# B&R Automation Studio project PO_automation
Automation Studio 4.5.2.102

## Configuration Config1

### Task classes (Cpu.sw)
```
Cyclic#1:
  Program <- Program.prg
Binaries: udbdef, TCData, ashwd, User, asfw, arconfig, sysconf, Role, ashwac, iomap
Libraries: library
```

## Logical view

Binary libraries used (declarations not repeated): operator, runtime, astime, AsIecCon

### Global.var
```iecst
VAR
	fb_controller : FB_Regulator;
	speed : REAL;
	counter : UINT;
	enable : BOOL;
	fb_motor2 : FB_Motor;
	fb_motor1 : FB_Motor;
END_VAR
```

### Library Logical/Libraries/library (ANSIC)

#### FB_Integrator.c
```c
#include <bur/plctypes.h>
#ifdef __cplusplus
	extern "C"
	{
#endif
	#include "library.h"
#ifdef __cplusplus
	};
#endif
/* TODO: Add your comment here */
void FB_Integrator(struct FB_Integrator* inst)
{
	/*TODO: Add your code here*/
	inst->out = inst->dt * inst->in + inst->prev_value;
	inst->prev_value = inst->out;
}
```

#### library.fun - Exported functions and function blocks
```iecst
{REDUND_ERROR} FUNCTION_BLOCK FB_Integrator (*TODO: Add your comment here*) (*$GROUP=User,$CAT=User,$GROUPICON=User.png,$CATICON=User.png*)
	VAR_INPUT
		in : {REDUND_UNREPLICABLE} REAL;
		dt : REAL;
	END_VAR
	VAR_OUTPUT
		out : {REDUND_UNREPLICABLE} REAL;
	END_VAR
	VAR
		prev_value : REAL;
	END_VAR
END_FUNCTION_BLOCK

{REDUND_ERROR} FUNCTION_BLOCK FB_Regulator (*TODO: Add your comment here*) (*$GROUP=User,$CAT=User,$GROUPICON=User.png,$CATICON=User.png*)
	VAR_INPUT
		e : {REDUND_UNREPLICABLE} REAL;
		dt : REAL;
	END_VAR
	VAR_OUTPUT
		u : {REDUND_UNREPLICABLE} REAL;
	END_VAR
	VAR
		k_p : {REDUND_UNREPLICABLE} REAL;
		k_i : {REDUND_UNREPLICABLE} REAL;
		integrator : {REDUND_UNREPLICABLE} FB_Integrator;
		iyOld : {REDUND_UNREPLICABLE} REAL;
		max_abs_value : {REDUND_UNREPLICABLE} REAL;
		ls : {REDUND_UNREPLICABLE} REAL;
		sum : {REDUND_UNREPLICABLE} REAL;
	END_VAR
END_FUNCTION_BLOCK

{REDUND_ERROR} FUNCTION_BLOCK FB_Motor (*TODO: Add your comment here*) (*$GROUP=User,$CAT=User,$GROUPICON=User.png,$CATICON=User.png*)
	VAR_INPUT
		u : REAL;
		dt : REAL;
	END_VAR
	VAR_OUTPUT
		w : REAL;
		phi : REAL;
	END_VAR
	VAR
		Tm : REAL;
		integrator : FB_Integrator;
		ke : REAL;
	END_VAR
END_FUNCTION_BLOCK
```

#### FB_Regulator.c
```c
#include <bur/plctypes.h>
#ifdef __cplusplus
	extern "C"
	{
#endif
	#include "library.h"
#ifdef __cplusplus
	};
#endif
/* TODO: Add your comment here */
void FB_Regulator(struct FB_Regulator* inst)
{
	inst->integrator.dt = inst->dt;

	REAL a = inst->e * inst->k_p;
	REAL b = inst->e * inst->k_i;

	a = a > inst->max_abs_value ? inst->max_abs_value : a;
	a = a < -inst->max_abs_value ? -inst->max_abs_value : a;

	inst->integrator.in = b + inst->ls;
	FB_Integrator(&inst->integrator);

	inst->sum = a + inst->integrator.out;
	inst->u = inst->sum;
	inst->u = inst->u > inst->max_abs_value ? inst->max_abs_value : inst->u;
	inst->u = inst->u < -inst->max_abs_value ? -inst->max_abs_value : inst->u;

	inst->ls = inst->u - inst->sum;
}
```

#### FB_Motor.c
```c
#include <bur/plctypes.h>
#ifdef __cplusplus
	extern "C"
	{
#endif
	#include "library.h"
#ifdef __cplusplus
	};
#endif
/* TODO: Add your comment here */
void FB_Motor(struct FB_Motor* inst)
{
	inst->integrator.dt = inst->dt;
	REAL a = inst->u / inst->ke - inst->w;
	REAL b = a / inst->Tm;

	inst->integrator.in = b;
	FB_Integrator(&inst->integrator);

	inst->w = inst->integrator.out;
}
```

### Program Logical/Program

#### Cyclic.c
```c
#include <bur/plctypes.h>

#ifdef _DEFAULT_INCLUDES
	#include <AsDefault.h>
#endif

void _CYCLIC ProgramCyclic(void)
{
	if(enable)
	{
		if(counter == 1000)
		{
			speed = 60;
		}
		if(counter == 1100)
		{
			speed = 0;
			counter = 0;
		}
		counter = counter + 1;

		fb_controller.e = speed - fb_motor1.w;
		FB_Regulator(&fb_controller);

		fb_motor1.u = fb_controller.u;
		FB_Motor(&fb_motor1);

		fb_motor2.u = speed * fb_motor2.ke;
		FB_Motor(&fb_motor2);

	}
}
```

#### Init.c
```c
#include <bur/plctypes.h>

#ifdef _DEFAULT_INCLUDES
	#include <AsDefault.h>
#endif

void _INIT ProgramInit(void)
{
	fb_motor1.dt = 0.02;
	fb_motor1.ke = 0.23;
	fb_motor1.Tm = 0.1;
	fb_motor1.u = 0;

	fb_motor2.dt = 0.02;
	fb_motor2.ke = 0.23;
	fb_motor2.Tm = 0.1;
	fb_motor2.u = 0;

	fb_controller.dt = 0.015;
	fb_controller.k_i = 4.9;
	fb_controller.k_p = 0.46;
	fb_controller.max_abs_value = 24.0;

	speed = 0;
	counter = 0;
	enable = 1;
}
```

Listed in the project but not available here: Logical/Libraries/library/Types.typ, Logical/Libraries/library/Constants.var
